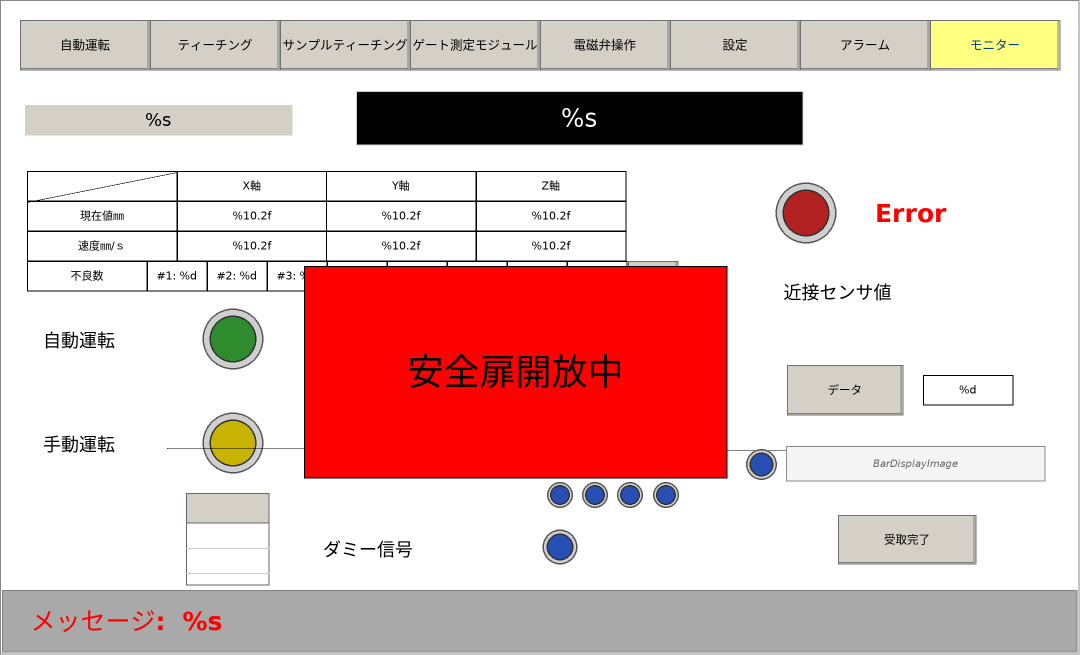
VISUALIZATION s_monitor  // 1080x655
    Rectangle (0,0 1080x655)
    Rectangle (177,201 150x30), "%10.2f", text variable: gvl_axis.axisX.NcToPlc.ActPos
    Rectangle (326,201 150x30), "%10.2f", text variable: gvl_axis.axisY.NcToPlc.ActPos
    Rectangle (476,201 150x30), "%10.2f", text variable: gvl_axis.axisZ.NcToPlc.ActPos
    Rectangle (177,171 150x30), "X軸"
    Rectangle (326,171 150x30), "Y軸"
    Rectangle (476,171 150x30), "Z軸"
    Rectangle (177,231 150x30), "%10.2f", text variable: gvl_axis.axisX.NcToPlc.ActVelo
    Rectangle (326,231 150x30), "%10.2f", text variable: gvl_axis.axisY.NcToPlc.ActVelo
    Rectangle (476,231 150x30), "%10.2f", text variable: gvl_axis.axisZ.NcToPlc.ActVelo
    Rectangle (27,171 150x30)
    Rectangle (27,201 150x30), "現在値㎜"
    Rectangle (27,231 150x30), "速度㎜/ｓ"
    Line (27,202) (177,172)
    Lamp1 (198,304 70x70), variable: gvl_param.var_currentMode = eP_programMode.auto, style: Lamp-Lamp1-Green
    Lamp1 (198,408 70x70), variable: gvl_param.var_currentMode = eP_programMode.manual, style: Lamp-Lamp1-Yellow
    Lamp1 (771,178 70x70), variable: gvl_param.var_currentMode = eP_programMode.error, invisible if: gvl_param.var_currentMode <> eP_programMode.error, style: Lamp-Lamp1-Red
    Label (839,194 144x38), "Error", invisible if: gvl_param.var_currentMode <> eP_programMode.error
    Line (167,448) (442,447)
    Line (560,451) (835,450)
    RoundedRectangle (25,105 267x30), "%s", text variable: gvl_visu.var_DT
    Rectangle (356,91 447x54), "%s", text variable: gvl_param.var_productInfo[gvl_param.var_currentProductID].name
    Button (628,261 50x30), "CLR"
        tap gvl_visu.flg_btn_clrDefectiveQty
    Rectangle (147,261 60x30), "#1: %d", text variable: gvl_auto.var_defectiveLens[1]
    Rectangle (267,261 60x30), "#3: %d", text variable: gvl_auto.var_defectiveLens[3]
    Rectangle (207,261 60x30), "#2: %d", text variable: gvl_auto.var_defectiveLens[2]
    Rectangle (327,261 60x30), "#4: %d", text variable: gvl_auto.var_defectiveLens[4]
    Rectangle (387,261 60x30), "#5: %d", text variable: gvl_auto.var_defectiveLens[5]
    Rectangle (447,261 60x30), "#6: %d", text variable: gvl_auto.var_defectiveLens[6]
    Rectangle (507,261 60x30), "#7: %d", text variable: gvl_auto.var_defectiveLens[7]
    Rectangle (567,261 60x30), "#8: %d", text variable: gvl_auto.var_defectiveLens[8]
    Rectangle (27,261 120x30), "不良数"
    Label (733,278 209x30), "近接センサ値"
    Rectangle (923,375 90x30), "%d", text variable: gvl_io.in_wire_gateLength
    Lamp1 (744,447 35x35), variable: gvl_auto.gateLengthIsPassed, style: Lamp-Lamp1-Blue
    Lamp1 (540,424 40x40), variable: gvl_IO.flg_gateLengthIsSuccessed, style: Lamp-Lamp1-Blue
    Lamp1 (540,370 40x40), variable: gvl_io.flg_lensSetDone, style: Lamp-Lamp1-Blue
    Lamp1 (545,480 30x30), variable: gvl_io.in_bitNumber3, style: Lamp-Lamp1-Blue
    Label (320,379 200x30), "レンズセット完了信号"
    Label (320,430 200x30), "ゲート測定OK信号"
    Rectangle (40,326 140x30), "自動運転", text variable: gvl_auto.cavNo
    Label (320,328 200x30), "レンズ要求信号"
    Lamp1 (540,323 40x40), variable: gvl_io.flg_requestLens, style: Lamp-Lamp1-Red
    Lamp1 (540,527 40x40), variable: gvl_io.flg_dummySiganl, style: Lamp-Lamp1-Blue
    Lamp1 (580,480 30x30), variable: gvl_io.flg_bitNumber2, style: Lamp-Lamp1-Blue
    Lamp1 (615,480 30x30), variable: gvl_io.flg_bitNumber1, style: Lamp-Lamp1-Blue
    Lamp1 (651,480 30x30), variable: gvl_io.flg_bitNumber0, style: Lamp-Lamp1-Blue
    Label (529,457 165x30), "4 3 2 1"
    Label (320,535 200x30), "ダミー信号"
    Table (186,493 83x92), data array: gvl_auto.pocketNo
        p3854506369: gvl_auto.pocketNo[INDEX]
    Button (20,20 130x50), "自動運転"
        OnMouseClick: change screen: s_auto
    Button (150,20 130x50), "ティーチング"
        OnMouseClick: change screen: s_teaching1
    Button (670,20 130x50), "設定"
        OnMouseClick: change screen: s_setting
    Button (540,20 130x50), "電磁弁操作"
        OnMouseClick: change screen: s_manual
    Button (410,20 130x50), "ゲート測定モジュール"
        OnMouseClick: change screen: s_gm_teaching
    Button (800,20 130x50), "アラーム", colour toggle: gvl_io.flg_signalTowerRed
        OnMouseClick: change screen: s_alarm
    Button (280,20 130x50), "サンプルティーチング"
        OnMouseClick: change screen: s_sample
    BarDisplayImage (786,446 259x35), value: gvl_visu.var_curenntGateData, style: BarDisplayImage-Gray, scale format: %.1f, scale 0..3
    Button (787,365 116x50), "データ"
        OnMouseClick: change screen: s_gateLengthData
    Rectangle (304,266 423x212), "安全扉開放中", text variable: gvl_io.flg_frontSaftyDoor or gvl_param.var_currentMode <> eP_programMode.auto, invisible if: gvl_io.flg_frontSaftyDoor or gvl_param.var_currentMode <> eP_programMode.auto
    Button (930,20 130x50), "モニター"
        OnMouseClick: change screen: s_monitor
    Rectangle (40,430 140x30), "手動運転", text variable: gvl_auto.cavNo
    Button (838,515 138x49), "受取完了", invisible if: gvl_debug.flg_debug_run = FALSE OR gvl_io.flg_requestLens = FALSE
        tap gvl_visu.flg_btn_lensSetDone
    Rectangle (2,590 1075x62), "メッセージ: %s", text variable: gvl_visu.var_msg
END_VISUALIZATION

(* stored: Version 1.1.0.1, ProductVersion 3.1.4024.11
   Visu s_monitor: Id {ac7e6fc2-74f6-43c5-bf04-70414cee429c} *)
